// TIA Portal project "Ürün Ayrıştırma" (V17)

(* hardware
DEVICE "S7-1200 station_1"  S7-1200 Station
   slot 0: "Rack_0"  S7-1200 Rack  Rack  V1.0
   slot 1: "BitirmeProjesi"  CPU 1214C DC/DC/DC  6ES7 214-1AG40-0XB0  V4.4
DEVICE "PC-System_1"  SIMATIC PC station
   slot 0: "SIMATIC PC station"  Rail  SIMATIC PC-Station  V1.0
      slot 125: "Stationmanager"  Station_Manager  V6.0.4
   slot 1: "HMI_RT_1"  WinCC RT Advanced  6AV2 104-0xxxx-xxxx  17.0.0.0
      slot 33792: "Computer interface"  Host interface
   slot 2: "IE general_1"  IE General  IE_CP  V8.2.0
      slot 1: "PROFINET interface"  IEGeneral.Interface.8.2.0
*)

// ===== PLC "BitirmeProjesi"  CPU 1214C DC/DC/DC =====

VAR_GLOBAL   // PLC tag table "Default tag table"
   "Üst Sensör" AT %I0.0 : Bool;
   "Alt Sensör" AT %I0.1 : Bool;
   "Metal Sensörü" AT %I0.2 : Bool;
   "Motor" AT %Q0.2 : Bool;
   "Büyük" AT %Q0.3 : Bool;
   "Küçük" AT %Q0.4 : Bool;
   "Metal" AT %Q0.5 : Bool;
   "Step1" AT %Q0.0 : Bool;
   "Step2" AT %Q0.1 : Bool;
   "Kırmızı" AT %Q0.6 : Bool;
   "Yeşil" AT %Q0.7 : Bool;
   "Mavi" AT %Q1.0 : Bool;
   "Start" AT %M0.0 : Bool;
   "Step Pozisyon" AT %MD100 : Real;
   "Step Hız" AT %MD104 : Real;
   "Stop" AT %M0.1 : Bool;
   "Boyut Start" AT %M0.2 : Bool;
   "Materyal Start" AT %M0.3 : Bool;
   "Görüntü Start" AT %M0.4 : Bool;
   "Motor Start" AT %M0.5 : Bool;
   "Boyut" AT %M0.6 : Bool;
   "Materyal" AT %M0.7 : Bool;
   "Görüntü" AT %M1.0 : Bool;
   "BStepSet" AT %M1.1 : Bool;
   "KStepSet" AT %M1.2 : Bool;
   "MStepSet" AT %M1.3 : Bool;
   "RedStepSet" AT %M1.4 : Bool;
   "GreenStepSet" AT %M1.5 : Bool;
   "BlueStepSet" AT %M1.6 : Bool;
   "Home Başlat" AT %M1.7 : Bool;
   "Kırmızı Ürün" AT %M2.0 : Bool;
   "Yeşil Ürün" AT %M2.1 : Bool;
   "Mavi Ürün" AT %M2.2 : Bool;
   "BIG" AT %M2.3 : Bool;
   "SMALL" AT %M2.4 : Bool;
   "ALLOY" AT %M2.5 : Bool;
   "RED" AT %M2.6 : Bool;
   "GREEN" AT %M2.7 : Bool;
   "BLUE" AT %M3.0 : Bool;
   "HandStart" AT %M20.0 : Bool;
   "Metal Olmayan" AT %M3.1 : Bool;
   "MOStepSet" AT %M3.2 : Bool;
   "NON-ALLOY" AT %M3.3 : Bool;
END_VAR

// folder: System blocks/Program resources

DATA_BLOCK "Üst"   // DB1
{ S7_Optimized_Access := 'TRUE' }
AUTHOR : Simatic
FAMILY : IEC
NAME : IEC_TMR
VERSION : 1.0
// stored: InstanceOfName IEC_TIMER
"IEC_TIMER"
BEGIN
END_DATA_BLOCK

DATA_BLOCK "Alt"   // DB2
{ S7_Optimized_Access := 'TRUE' }
AUTHOR : Simatic
FAMILY : IEC
NAME : IEC_TMR
VERSION : 1.0
// stored: InstanceOfName IEC_TIMER
"IEC_TIMER"
BEGIN
END_DATA_BLOCK

DATA_BLOCK "BStepKapa"   // DB3
{ S7_Optimized_Access := 'TRUE' }
AUTHOR : Simatic
FAMILY : IEC
NAME : IEC_TMR
VERSION : 1.0
// stored: InstanceOfName IEC_TIMER
"IEC_TIMER"
BEGIN
END_DATA_BLOCK

DATA_BLOCK "KStepKapa"   // DB5
{ S7_Optimized_Access := 'TRUE' }
AUTHOR : Simatic
FAMILY : IEC
NAME : IEC_TMR
VERSION : 1.0
// stored: InstanceOfName IEC_TIMER
"IEC_TIMER"
BEGIN
END_DATA_BLOCK

DATA_BLOCK "Metal Zaman"   // DB6
{ S7_Optimized_Access := 'TRUE' }
AUTHOR : Simatic
FAMILY : IEC
NAME : IEC_TMR
VERSION : 1.0
// stored: InstanceOfName IEC_TIMER
"IEC_TIMER"
BEGIN
END_DATA_BLOCK

DATA_BLOCK "MStepKapa"   // DB7
{ S7_Optimized_Access := 'TRUE' }
AUTHOR : Simatic
FAMILY : IEC
NAME : IEC_TMR
VERSION : 1.0
// stored: InstanceOfName IEC_TIMER
"IEC_TIMER"
BEGIN
END_DATA_BLOCK

DATA_BLOCK "Kırmızı Süre"   // DB8
{ S7_Optimized_Access := 'TRUE' }
AUTHOR : Simatic
FAMILY : IEC
NAME : IEC_TMR
VERSION : 1.0
// stored: InstanceOfName IEC_TIMER
"IEC_TIMER"
BEGIN
END_DATA_BLOCK

DATA_BLOCK "Yeşil Süre"   // DB9
{ S7_Optimized_Access := 'TRUE' }
AUTHOR : Simatic
FAMILY : IEC
NAME : IEC_TMR
VERSION : 1.0
// stored: InstanceOfName IEC_TIMER
"IEC_TIMER"
BEGIN
END_DATA_BLOCK

DATA_BLOCK "Mavi Süre"   // DB10
{ S7_Optimized_Access := 'TRUE' }
AUTHOR : Simatic
FAMILY : IEC
NAME : IEC_TMR
VERSION : 1.0
// stored: InstanceOfName IEC_TIMER
"IEC_TIMER"
BEGIN
END_DATA_BLOCK

DATA_BLOCK "RedStepKapa"   // DB11
{ S7_Optimized_Access := 'TRUE' }
AUTHOR : Simatic
FAMILY : IEC
NAME : IEC_TMR
VERSION : 1.0
// stored: InstanceOfName IEC_TIMER
"IEC_TIMER"
BEGIN
END_DATA_BLOCK

DATA_BLOCK "GreenStepKapa"   // DB12
{ S7_Optimized_Access := 'TRUE' }
AUTHOR : Simatic
FAMILY : IEC
NAME : IEC_TMR
VERSION : 1.0
// stored: InstanceOfName IEC_TIMER
"IEC_TIMER"
BEGIN
END_DATA_BLOCK

DATA_BLOCK "BlueStepKapa"   // DB13
{ S7_Optimized_Access := 'TRUE' }
AUTHOR : Simatic
FAMILY : IEC
NAME : IEC_TMR
VERSION : 1.0
// stored: InstanceOfName IEC_TIMER
"IEC_TIMER"
BEGIN
END_DATA_BLOCK

DATA_BLOCK "Metal Olmayan Zaman"   // DB17
{ S7_Optimized_Access := 'TRUE' }
AUTHOR : Simatic
FAMILY : IEC
NAME : IEC_TMR
VERSION : 1.0
// stored: InstanceOfName IEC_TIMER
"IEC_TIMER"
BEGIN
END_DATA_BLOCK

DATA_BLOCK "MOStepKapa"   // DB18
{ S7_Optimized_Access := 'TRUE' }
AUTHOR : Simatic
FAMILY : IEC
NAME : IEC_TMR
VERSION : 1.0
// stored: InstanceOfName IEC_TIMER
"IEC_TIMER"
BEGIN
END_DATA_BLOCK

// folder: (top level)

DATA_BLOCK "Step Motor"   // DB4, Motion_DB
{ S7_Optimized_Access := 'TRUE' }
AUTHOR : SIMATIC
FAMILY : BasicMC
NAME : TO_PosAx
VERSION : 7.0
// stored: InstanceOfName TO_PositioningAxis
"TO_PositioningAxis"
BEGIN
   // Axis.LengthUnitNormalized.Distance = 1005
   // Axis.LengthUnit.LastDistance = 1005
   // Axis.DirectionOutputEnabledCU = TRUE
   // Axis.OnlinePtoModeCU = 16#0000_0002
   // Axis.SelectedChannel2EnumCU = %Q0.1
   // Axis.SelectedChannel1EnumCU = %Q0.0
   // Pulse.MinDeltaDeltaFrequencyCU = 0.004
   // Pulse.MaxDeltaDeltaFrequencyCU = 1.0E+10
   // Pulse.MinDeltaFrequencyCU = 0.005
   // Pulse.MaxDeltaFrequencyCU = 9.5E+9
   // Pulse.MinFrequencyCU = 1.0
   // Pulse.MaxFrequencyCU = 100000.0
   // Pulse.OutputSourceCU = 16#0000_0000
   // Axis.SelectPTO = 0
END_DATA_BLOCK

ORGANIZATION_BLOCK "Main"   // OB1, LAD, ProgramCycle
TITLE = "Main Program Sweep (Cycle)"
{ S7_Optimized_Access := 'TRUE' }
VERSION : 0.1
   VAR_INPUT
      Initial_Call : Bool;   // Initial call of this OB
      Remanence : Bool;   // =True, if remanent data are available
   END_VAR
BEGIN

REGION Network 1: Motor Başlat
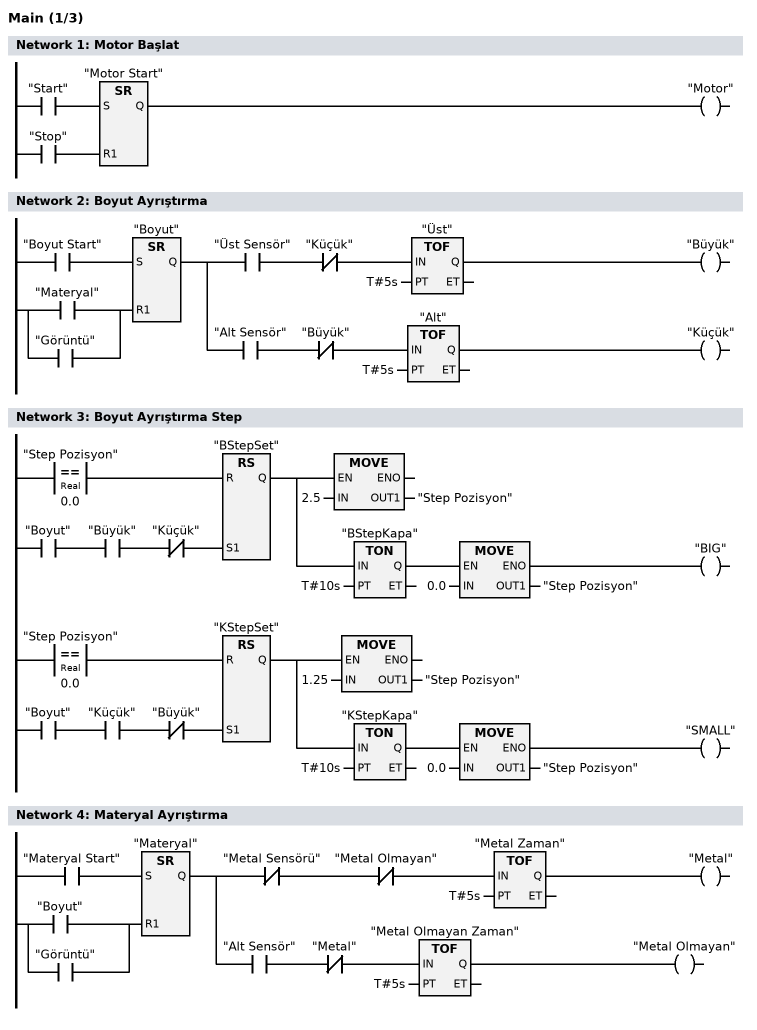
   RUNG wire#powerrail
      Contact( "Start" )
      S_SR(operand := "Motor Start", r1 := wire#w1)
      Coil( "Motor" )
   END_RUNG
   RUNG wire#powerrail
      Contact( "Stop" )
   END_RUNG wire#w1
   // the same network as SCL:
   IF "Start" THEN
       "Motor Start" := TRUE;   // SR flip-flop
   END_IF;
   IF "Stop" THEN "Motor Start" := FALSE; END_IF;
   "Motor" := "Motor Start";
END_REGION

REGION Network 2: Boyut Ayrıştırma
   IF "Boyut Start" THEN
       "Boyut" := TRUE;   // SR flip-flop
   END_IF;
   IF "Materyal" OR "Görüntü" THEN "Boyut" := FALSE; END_IF;
   "Üst".TOF(IN := "Boyut" AND "Üst Sensör" AND NOT "Küçük", PT := T#5s);
   "Büyük" := "Üst".Q;
   "Alt".TOF(IN := "Boyut" AND "Alt Sensör" AND NOT "Büyük", PT := T#5s);
   "Küçük" := "Alt".Q;
END_REGION

REGION Network 3: Boyut Ayrıştırma Step
   IF "Step Pozisyon" = 0.0 THEN
       "BStepSet" := FALSE;   // RS flip-flop
   END_IF;
   IF "Boyut" AND "Büyük" AND NOT "Küçük" THEN "BStepSet" := TRUE; END_IF;
   IF "BStepSet" THEN "Step Pozisyon" := 2.5; END_IF;
   "BStepKapa".TON(IN := "BStepSet", PT := T#10s);
   IF "BStepKapa".Q THEN "Step Pozisyon" := 0.0; END_IF;
   "BIG" := "BStepKapa".Q;
   IF "Step Pozisyon" = 0.0 THEN
       "KStepSet" := FALSE;   // RS flip-flop
   END_IF;
   IF "Boyut" AND "Küçük" AND NOT "Büyük" THEN "KStepSet" := TRUE; END_IF;
   IF "KStepSet" THEN "Step Pozisyon" := 1.25; END_IF;
   "KStepKapa".TON(IN := "KStepSet", PT := T#10s);
   IF "KStepKapa".Q THEN "Step Pozisyon" := 0.0; END_IF;
   "SMALL" := "KStepKapa".Q;
END_REGION

REGION Network 4: Materyal Ayrıştırma
   IF "Materyal Start" THEN
       "Materyal" := TRUE;   // SR flip-flop
   END_IF;
   IF "Boyut" OR "Görüntü" THEN "Materyal" := FALSE; END_IF;
   "Metal Zaman".TOF(IN := "Materyal" AND NOT "Metal Sensörü" AND NOT "Metal Olmayan", PT := T#5s);
   "Metal" := "Metal Zaman".Q;
   "Metal Olmayan Zaman".TOF(IN := "Materyal" AND "Alt Sensör" AND NOT "Metal", PT := T#5s);
   "Metal Olmayan" := "Metal Olmayan Zaman".Q;
END_REGION

REGION Network 5: Materyal Ayrıştırma Step
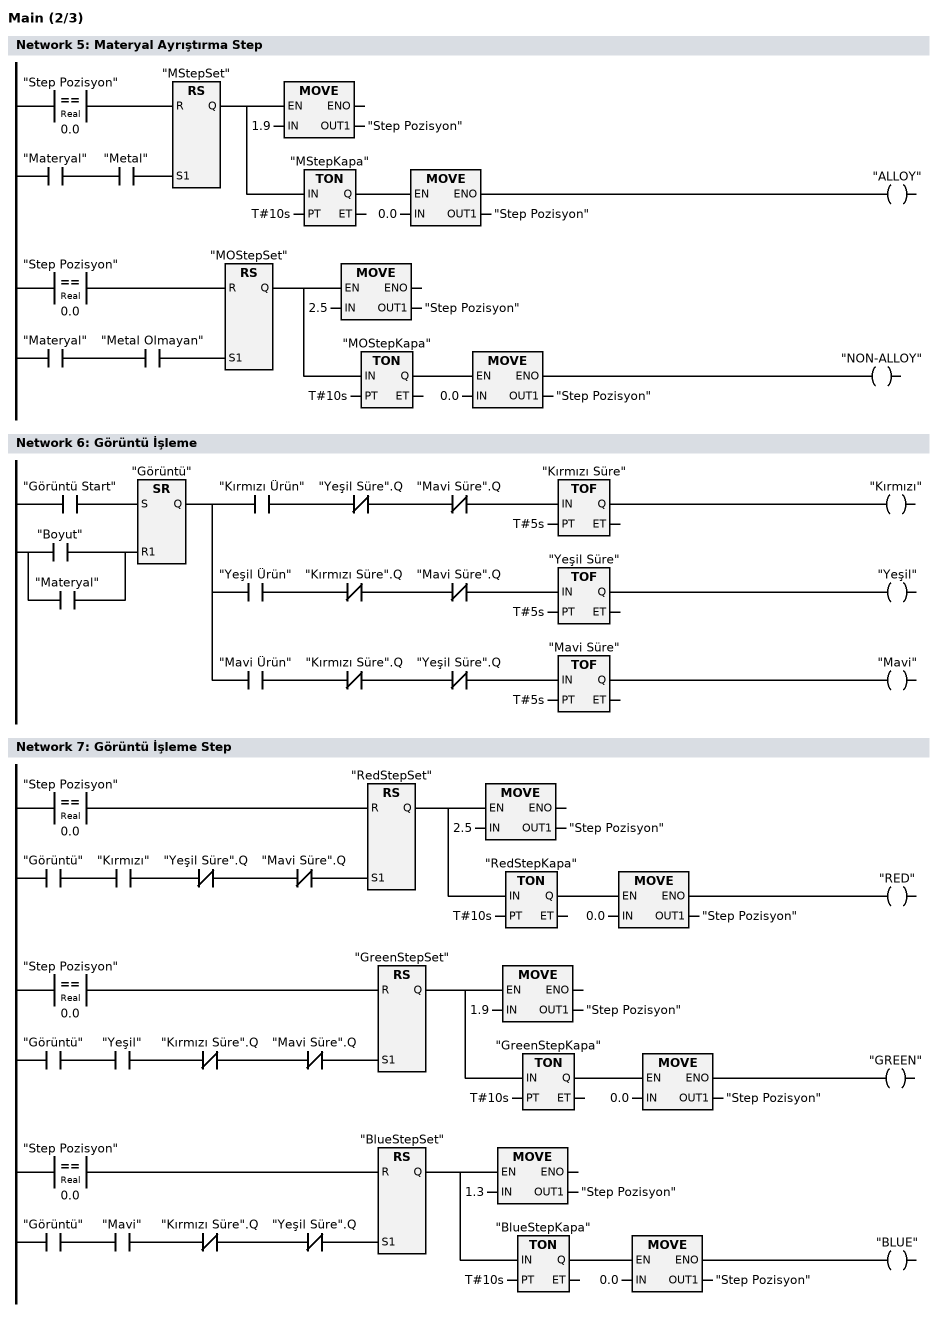
   IF "Step Pozisyon" = 0.0 THEN
       "MStepSet" := FALSE;   // RS flip-flop
   END_IF;
   IF "Materyal" AND "Metal" THEN "MStepSet" := TRUE; END_IF;
   IF "MStepSet" THEN "Step Pozisyon" := 1.9; END_IF;
   "MStepKapa".TON(IN := "MStepSet", PT := T#10s);
   IF "MStepKapa".Q THEN "Step Pozisyon" := 0.0; END_IF;
   "ALLOY" := "MStepKapa".Q;
   IF "Step Pozisyon" = 0.0 THEN
       "MOStepSet" := FALSE;   // RS flip-flop
   END_IF;
   IF "Materyal" AND "Metal Olmayan" THEN "MOStepSet" := TRUE; END_IF;
   IF "MOStepSet" THEN "Step Pozisyon" := 2.5; END_IF;
   "MOStepKapa".TON(IN := "MOStepSet", PT := T#10s);
   IF "MOStepKapa".Q THEN "Step Pozisyon" := 0.0; END_IF;
   "NON-ALLOY" := "MOStepKapa".Q;
END_REGION

REGION Network 6: Görüntü İşleme
   IF "Görüntü Start" THEN
       "Görüntü" := TRUE;   // SR flip-flop
   END_IF;
   IF "Boyut" OR "Materyal" THEN "Görüntü" := FALSE; END_IF;
   "Kırmızı Süre".TOF(IN := "Görüntü" AND "Kırmızı Ürün" AND NOT "Yeşil Süre".Q AND NOT "Mavi Süre".Q,
                      PT := T#5s);
   "Kırmızı" := "Kırmızı Süre".Q;
   "Yeşil Süre".TOF(IN := "Görüntü" AND "Yeşil Ürün" AND NOT "Kırmızı Süre".Q AND NOT "Mavi Süre".Q, PT := T#5s);
   "Yeşil" := "Yeşil Süre".Q;
   "Mavi Süre".TOF(IN := "Görüntü" AND "Mavi Ürün" AND NOT "Kırmızı Süre".Q AND NOT "Yeşil Süre".Q, PT := T#5s);
   "Mavi" := "Mavi Süre".Q;
END_REGION

REGION Network 7: Görüntü İşleme Step
   IF "Step Pozisyon" = 0.0 THEN
       "RedStepSet" := FALSE;   // RS flip-flop
   END_IF;
   IF "Görüntü" AND "Kırmızı" AND NOT "Yeşil Süre".Q AND NOT "Mavi Süre".Q THEN "RedStepSet" := TRUE; END_IF;
   IF "RedStepSet" THEN "Step Pozisyon" := 2.5; END_IF;
   "RedStepKapa".TON(IN := "RedStepSet", PT := T#10s);
   IF "RedStepKapa".Q THEN "Step Pozisyon" := 0.0; END_IF;
   "RED" := "RedStepKapa".Q;
   IF "Step Pozisyon" = 0.0 THEN
       "GreenStepSet" := FALSE;   // RS flip-flop
   END_IF;
   IF "Görüntü" AND "Yeşil" AND NOT "Kırmızı Süre".Q AND NOT "Mavi Süre".Q THEN
       "GreenStepSet" := TRUE;
   END_IF;
   IF "GreenStepSet" THEN "Step Pozisyon" := 1.9; END_IF;
   "GreenStepKapa".TON(IN := "GreenStepSet", PT := T#10s);
   IF "GreenStepKapa".Q THEN "Step Pozisyon" := 0.0; END_IF;
   "GREEN" := "GreenStepKapa".Q;
   IF "Step Pozisyon" = 0.0 THEN
       "BlueStepSet" := FALSE;   // RS flip-flop
   END_IF;
   IF "Görüntü" AND "Mavi" AND NOT "Kırmızı Süre".Q AND NOT "Yeşil Süre".Q THEN
       "BlueStepSet" := TRUE;
   END_IF;
   IF "BlueStepSet" THEN "Step Pozisyon" := 1.3; END_IF;
   "BlueStepKapa".TON(IN := "BlueStepSet", PT := T#10s);
   IF "BlueStepKapa".Q THEN "Step Pozisyon" := 0.0; END_IF;
   "BLUE" := "BlueStepKapa".Q;
END_REGION

REGION Network 8: SCADA Home Butonu Ekle
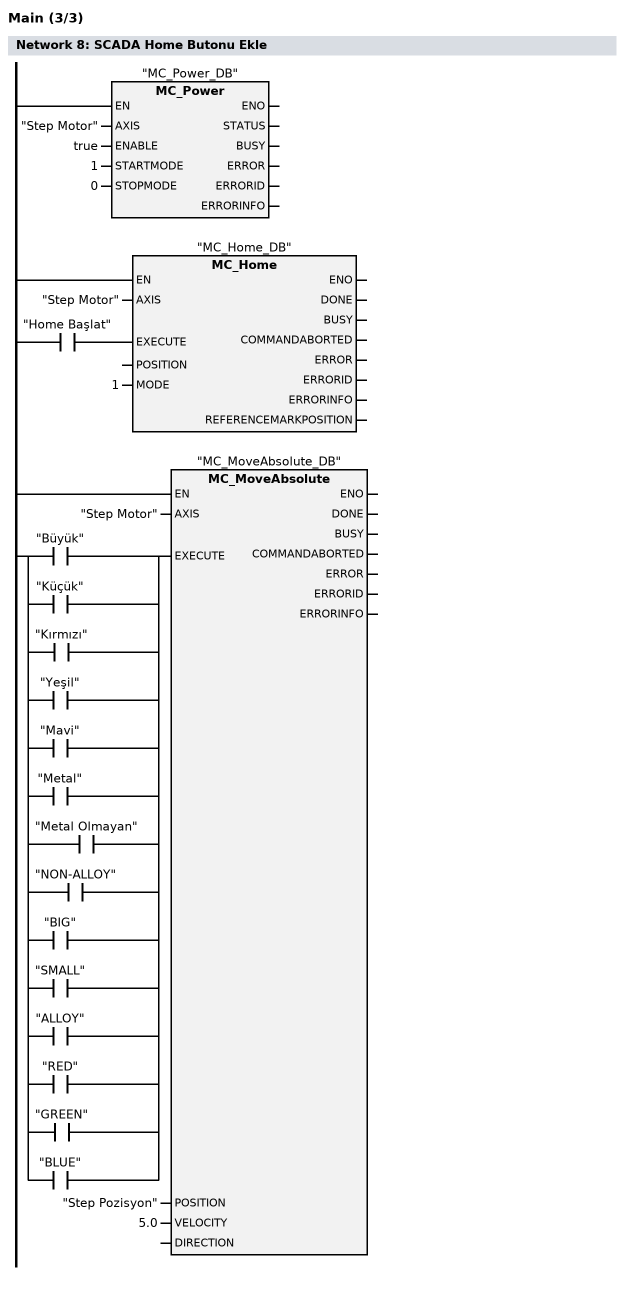
   "MC_Power_DB"(Axis := "Step Motor", Enable := true, StartMode := 1, StopMode := 0);   // MC_Power
   "MC_Home_DB"(Axis := "Step Motor", Execute := "Home Başlat", Mode := 1);   // MC_Home
   "MC_MoveAbsolute_DB"(Axis := "Step Motor",   // MC_MoveAbsolute
                        Execute := "Büyük" OR "Küçük" OR "Kırmızı" OR "Yeşil" OR "Mavi" OR "Metal" OR "Metal Olmayan" OR "NON-ALLOY" OR "BIG" OR "SMALL" OR "ALLOY" OR "RED" OR "GREEN" OR "BLUE",
                        Position := "Step Pozisyon",
                        Velocity := 5.0);
END_REGION
END_ORGANIZATION_BLOCK

(* ===== HMI "HMI_RT_1" =====
system functions are stored by id; their names below are inferred from use
connection "HMI_Connection_1": ETHERNET, S7_1200_OMS

HMI tags "Default tag table"
   "Start" : Bool = PLC Start AT %M0.0, 1 s
   "Stop" : Bool = PLC Stop AT %M0.1, 1 s

screen "Screen_1" 1024x768
   Button "Button_1" at 261,145 size 72x70; TextOff 'Start'
      on Click: SetBit("Start")
      on Press: SetBit("Start")
      on Release: ResetBit("Start")
   Button "Button_2" at 367,141 size 85x74; TextOff 'Stop'
      on Click: SetBit("Stop")
      on Press: ResetBit("Stop")
      on Release: ResetBit("Stop")
*)